// TIA Portal V17 export
// export: Created 2022-07-20T07:02:38.0991787Z, ExportSetting WithDefaults, DisplayName Totally Integrated Automation Portal, DisplayVersion V17, DisplayName TIA Portal Openness, DisplayVersion V17, DisplayName TIA Portal Version Control Interface, DisplayVersion V17, DisplayName SINAMICS Startdrive Advanced, DisplayVersion V17, DisplayName SINAMICS Startdrive G130, G150, S120, S150, SINAMICS MV, S210, DisplayVersion V17, DisplayName SINAMICS Startdrive G110M, G120, G120C, G120D, G120P, G115D, DisplayVersion V17, DisplayName STEP 7 Professional, DisplayVersion V17, DisplayName STEP 7 Safety, DisplayVersion V17, DisplayName WinCC Advanced, DisplayVersion V17
VAR_GLOBAL   // PLC tag table "IFM_IO_CommunicationTable"
   IFM_IO_AL2301_IN_Byte0 AT %IB873 : Byte;
   IFM_IO_AL2301_IN_Byte1 AT %IB874 : Byte;
   IFM_IO_AL2301_IN_Byte2 AT %IB875 : Byte;
   IFM_IO_AL2301_IN_Byte3 AT %IB876 : Byte;
   IFM_IO_AL2301_IN_Byte4 AT %IB877 : Byte;
   IFM_IO_AL2301_IN_Byte5 AT %IB878 : Byte;
   IFM_IO_AL2301_IN_Byte6 AT %IB879 : Byte;
   IFM_IO_AL2301_IN_Byte7 AT %IB880 : Byte;
   IFM_IO_AL2301_IN_Byte8 AT %IB881 : Byte;
   IFM_IO_AL2301_IN_Byte9 AT %IB882 : Byte;
   IFM_IO_AL2301_IN_Byte10 AT %IB883 : Byte;
   IFM_IO_AL2301_IN_Byte11 AT %IB884 : Byte;
   IFM_IO_AL2301_IN_Byte12 AT %IB885 : Byte;
   IFM_IO_AL2301_IN_Byte13 AT %IB886 : Byte;
   IFM_IO_AL2301_IN_Byte14 AT %IB887 : Byte;
   IFM_IO_AL2301_IN_Byte15 AT %IB888 : Byte;
   IFM_IO_AL2301_IN_Byte16 AT %IB889 : Byte;
   IFM_IO_AL2301_IN_Byte17 AT %IB890 : Byte;
   IFM_IO_AL2301_IN_Byte18 AT %IB891 : Byte;
   IFM_IO_AL2301_IN_Byte19 AT %IB892 : Byte;
   IFM_IO_AL2301_IN_Byte20 AT %IB893 : Byte;
   IFM_IO_AL2301_IN_Byte21 AT %IB894 : Byte;
   IFM_IO_AL2301_IN_Byte22 AT %IB895 : Byte;
   IFM_IO_AL2301_IN_Byte23 AT %IB896 : Byte;
   IFM_IO_AL2301_IN_Byte24 AT %IB897 : Byte;
   IFM_IO_AL2301_IN_Byte25 AT %IB898 : Byte;
   IFM_IO_AL2301_IN_Byte26 AT %IB899 : Byte;
   IFM_IO_AL2301_IN_Byte27 AT %IB900 : Byte;
   IFM_IO_AL2301_IN_Byte28 AT %IB901 : Byte;
   IFM_IO_AL2301_IN_Byte29 AT %IB902 : Byte;
   IFM_IO_AL2301_IN_Byte30 AT %IB903 : Byte;
   IFM_IO_AL2301_IN_Byte31 AT %IB904 : Byte;
   IFM_IO_AL2301_OUT_Byte0 AT %QB834 : Byte;
   IFM_IO_AL2301_OUT_Byte1 AT %QB835 : Byte;
   IFM_IO_AL2301_OUT_Byte2 AT %QB836 : Byte;
   IFM_IO_AL2301_OUT_Byte3 AT %QB837 : Byte;
   IFM_IO_AL2301_OUT_Byte4 AT %QB838 : Byte;
   IFM_IO_AL2301_OUT_Byte5 AT %QB839 : Byte;
   IFM_IO_AL2301_OUT_Byte6 AT %QB840 : Byte;
   IFM_IO_AL2301_OUT_Byte7 AT %QB841 : Byte;
   IFM_IO_AL2301_OUT_Byte8 AT %QB842 : Byte;
   IFM_IO_AL2301_OUT_Byte9 AT %QB843 : Byte;
   IFM_IO_AL2301_OUT_Byte10 AT %QB844 : Byte;
   IFM_IO_AL2301_OUT_Byte11 AT %QB845 : Byte;
   IFM_IO_AL2301_OUT_Byte12 AT %QB846 : Byte;
   IFM_IO_AL2301_OUT_Byte13 AT %QB847 : Byte;
   IFM_IO_AL2301_OUT_Byte14 AT %QB848 : Byte;
   IFM_IO_AL2301_OUT_Byte15 AT %QB849 : Byte;
   IFM_IO_AL2301_OUT_Byte16 AT %QB850 : Byte;
   IFM_IO_AL2301_OUT_Byte17 AT %QB851 : Byte;
   IFM_IO_AL2301_OUT_Byte18 AT %QB852 : Byte;
   IFM_IO_AL2301_OUT_Byte19 AT %QB853 : Byte;
   IFM_IO_AL2301_OUT_Byte20 AT %QB854 : Byte;
   IFM_IO_AL2301_OUT_Byte21 AT %QB855 : Byte;
   IFM_IO_AL2301_OUT_Byte22 AT %QB856 : Byte;
   IFM_IO_AL2301_OUT_Byte23 AT %QB857 : Byte;
   IFM_IO_AL2301_OUT_Byte24 AT %QB858 : Byte;
   IFM_IO_AL2301_OUT_Byte25 AT %QB859 : Byte;
   IFM_IO_AL2301_OUT_Byte26 AT %QB860 : Byte;
   IFM_IO_AL2301_OUT_Byte27 AT %QB861 : Byte;
   IFM_IO_AL2301_OUT_Byte28 AT %QB862 : Byte;
   IFM_IO_AL2301_OUT_Byte29 AT %QB863 : Byte;
   IFM_IO_AL2301_OUT_Byte30 AT %QB864 : Byte;
   IFM_IO_AL2301_OUT_Byte31 AT %QB865 : Byte;
END_VAR
